// TwinCAT 3 PLC project PLC
// ProgramVersion: 3.1.4026.13
// libraries:
//   Tc2_Standard, * (Beckhoff Automation GmbH)
//   Tc2_System, * (Beckhoff Automation GmbH)
//   Tc3_Module, * (Beckhoff Automation GmbH)
// project tree:
//   Control/ FB_ControlSignal.TcPOU, FB_FeedForward.TcPOU, FB_PID.TcPOU (not stored), FB_Running.TcPOU (not stored), G_Mode.TcGVL
//   Filtering/ FB_Filtering.TcPOU (not stored), G_Filtered.TcGVL (not stored)
//   GVL/ G_Enables.TcGVL (not stored), G_FilterConstants.TcGVL (not stored), G_OPC.TcGVL, G_Parameter.TcGVL
//   Inputs/Function Blocks/ FB_FlowTransform.TcPOU, FB_JoystickInputScaling.TcPOU, FB_Normalize.TcPOU (not stored), FB_Normalize_Joystick.TcPOU, FB_PositionInputScaling.TcPOU (not stored)
//   Inputs/ G_Inputs.TcGVL
//   MotionRef/ FB_AutoClock.TcPOU (not stored), FB_DeadbandTester.TcPOU, FB_InitialPos.TcPOU (not stored), FB_MotionRef.TcPOU, FB_RunClock.TcPOU (not stored)
//   Outputs/ FB_ValveOutput.TcPOU (not stored), G_Output.TcGVL (not stored)
//   / PlcTask.TcTTO (not stored)
//   Programs/ MAIN.TcPOU (not stored), P_ControlBlock.TcPOU, P_FeedForward.TcPOU (not stored), P_Filtering.TcPOU (not stored), P_Inputs.TcPOU, P_Modes.TcPOU (not stored), P_Output.TcPOU (not stored), P_PID.TcPOU (not stored), P_RunClock.TcPOU (not stored)
//   XML/ FB_Derivator.TcPOU (not stored), FB_Integrator.TcPOU (not stored), G_Init.TcGVL (not stored)
// real-time tasks:
//   TASK PlcTask: cycle T#1ms, priority 20, ADS port 350
// I/O:
//   DEVICE Device 4 (EtherCAT), AmsNetId 5.107.189.26.5.1
//     RIO (EK1100) [EK1100 EtherCAT Coupler (2A E-Bus)]
//       DI (EL1008) [EL1008 8Ch. Dig. Input 24V, 3ms]
//       DO (EL2008) [EL2008 8Ch. Dig. Output 24V, 0.5A]
//       AI1 (EL3068) [EL3068 8Ch. Ana. Input 0-10V]
//       AI2 (EL3068) [EL3068 8Ch. Ana. Input 0-10V]
//       AI3 (EL3174) [EL3174 4Ch. Ana. Input +/-10V Diff., +/-20mA SingleEnded, 16 Bit]
//       AO (EL4104) [EL4104 4Ch. Ana. Output 0-10V, 16bit]
//       End Cap (EL9011) [EL9011 End Terminal]
// variable links:
//   PLC/PLC Instance <-> Device 4 (EtherCAT)/RIO (EK1100)/AI1 (EL3068)
//     PlcTask Inputs/G_Inputs.nRawJoystick <-> AI Standard Channel 2/Value
//     PlcTask Inputs/G_Inputs.nRawPistonPosition <-> AI Standard Channel 3/Value
//   PLC/PLC Instance <-> Device 4 (EtherCAT)/RIO (EK1100)/AI2 (EL3068)
//     PlcTask Inputs/G_Inputs.nRawPa <-> AI Standard Channel 4/Value
//     PlcTask Inputs/G_Inputs.nRawPaLower <-> AI Standard Channel 5/Value
//     PlcTask Inputs/G_Inputs.nRawPb <-> AI Standard Channel 6/Value
//     PlcTask Inputs/G_Inputs.nRawPs <-> AI Standard Channel 1/Value
//   PLC/PLC Instance <-> Device 4 (EtherCAT)/RIO (EK1100)/AI3 (EL3174)
//     PlcTask Inputs/G_Inputs.nRawFlow <-> AI Standard Channel 1/Value
//   PLC/PLC Instance <-> Device 4 (EtherCAT)/RIO (EK1100)/AO (EL4104)
//     PlcTask Outputs/G_Output.nValveOutput <-> AO Output Channel 1/Analog output
//   PLC/PLC Instance <-> Device 4 (EtherCAT)/RIO (EK1100)/DI (EL1008)
//     PlcTask Inputs/G_Inputs.bAuto <-> Channel 1/Input
//     PlcTask Inputs/G_Inputs.bManual <-> Channel 2/Input
//     PlcTask Inputs/G_Inputs.bStartButton <-> Channel 3/Input
//     PlcTask Inputs/G_Inputs.bStopButton <-> Channel 4/Input
//   PLC/PLC Instance <-> Device 4 (EtherCAT)/RIO (EK1100)/DO (EL2008)
//     PlcTask Outputs/G_Output.bGreenLight <-> Channel 1/Output
//     PlcTask Outputs/G_Output.bRedLight <-> Channel 2/Output
//     PlcTask Outputs/G_Output.bRunning <-> Channel 3/Output

// ---- Control/G_Mode.TcGVL
{attribute 'qualified_only'}
VAR_GLOBAL
	bRunning : BOOL;
	bManual : BOOL;
	bAuto : BOOL;
END_VAR

// ---- GVL/G_OPC.TcGVL
{attribute 'qualified_only'}
VAR_GLOBAL
	
	// Unfiltered Pressures
	fPa : LREAL;
	fPb : LREAL;
	fPs : LREAL;
	fPaLower : LREAL;
	
	// Filtered Pressures
	fPaFiltered : LREAL;
	fPbFiltered : LREAL;
	fPsFiltered : LREAL;
	fPaLowerFiltered : LREAL;
	
	
	fPistonPosition : LREAL;
	fJoystick : LREAL;
	fFlow : LREAL;
	fFlowBit : LREAL;
	
	fXRef : LREAL;
	fXDotRef : LREAL;
	
	fU : LREAL;
	fTime : LREAL;
	fError : LREAL;
	fSignalPID : LREAL;
	fUFF : LREAL;
END_VAR

// ---- GVL/G_Parameter.TcGVL
{attribute 'qualified_only'}
VAR_GLOBAL
	// Motion Ref
	fAmplitude : LREAL := 0.1;
	fMean : LREAL := 0.2;
	fFrequency : LREAL := 0.05;
	
	fQMaxDown : LREAL := 15.9;
	fQMaxUp : LREAL := 24.4;
	fDeadUp : LREAL := 0.13;
	fDeadDown : LREAL := 0.12;
	
	// Deadband test
	fConst : LREAL := 0.0; // [-1, 1]

	
	fCycleTime : LREAL := 0.001; // Time Step [s]
	fQConst : LREAL := 15;
	
	// PID-constants
	Kp 	: LREAL := 7.0; // P
	Ki 	: LREAL := 0.0;	// I
	Kd 	: LREAL := 0.0;	// D
	KFF : LREAL := 0.85; // Coefficient of FeedForward
	
END_VAR

// ---- Inputs/G_Inputs.TcGVL
{attribute 'qualified_only'}
VAR_GLOBAL
	// Mode Selector
	bManual 			AT %I* : BOOL;
	bAuto	 			AT %I* : BOOL;
	bStartButton		AT %I* : BOOL;
	bStopButton			AT %I* : BOOL;
	
	// Raw Pressure Values
	nRawPa 				AT %I*	: INT;
	nRawPb				AT %I*	: INT;
	nRawPs				AT %I*	: INT;
	nRawPaLower			AT %I* 	: INT;
	
	// Raw Position Values
	nRawPistonPosition 	AT %I*	: INT;
	nRawJoystick		AT %I*	: INT;
	nRawFlow			AT %I*	: INT; // [-150, 150]
END_VAR

// ---- Control/FB_ControlSignal.TcPOU
FUNCTION_BLOCK FB_ControlSignal
VAR_INPUT
	fUFF : LREAL;
	fPID : LREAL;
	bEnableU : BOOL;
	fQMaxUp 	: LREAL; // Needs to be positive (22)
	fQMaxDown 	: LREAL; // Needs to be positive (15)
	fDeadUp		: LREAL; // Needs to be positive (0.155)
	fDeadDown 	: LREAL; // Needs to be positive (0.18)
	
	fXDotRef	: LREAL;
	fError		: LREAL;
END_VAR
VAR_OUTPUT
	fU : LREAL;
END_VAR
VAR

	fUTemp : LREAL;
	fUTemp2 : LREAL;
	fUMax : LREAL := 0.9;
END_VAR

IF bEnableU THEN
	fUTemp := fUFF  - fPID;
	
	// Deadband compensation
	IF (fXDotRef > 0 OR fXDotRef < 0) OR fError > 0.002 THEN
		IF fUTemp <= 0.0 THEN	// Upwards
			fUTemp2 := fUTemp - fDeadUp;
		ELSIF fUTemp > 0.0 THEN // Downwards
			fUTemp2 := fUTemp + fDeadDown;
		END_IF
		
		IF fUTemp2 >= fUMax THEN
			fU := fUMax;
		ELSIF fUTemp2 <= -fUMax THEN
			fU := -fUMax;
		ELSE
			fU := fUTemp2;
		END_IF
	ELSE
		fU := 0.0;
	END_IF
END_IF

END_FUNCTION_BLOCK

// ---- Control/FB_FeedForward.TcPOU
FUNCTION_BLOCK FB_FeedForward
VAR_INPUT
	fXDotRef 	: LREAL; // Motion Referance
	fQMaxUp 	: LREAL; // Needs to be positive (22)
	fQMaxDown 	: LREAL; // Needs to be positive (15)
	fDeadUp		: LREAL; // Needs to be positive (0.155)
	fDeadDown 	: LREAL; // Needs to be positive (0.18)
	fPs 		: LREAL;
	fPa			: LREAL;
	fPb			: LREAL;
	fKFF 		: LREAL; // Coefficient of FeedForward
END_VAR
VAR_OUTPUT
	fUFF : LREAL;
END_VAR
VAR
	fUTemp : LREAL;
	fUMax : LREAL := 0.9;
	fQRef : LREAL;
	fAp : LREAL := 33.1 / 10000.0;
	fAa : LREAL := 23.56 / 10000.0;
	
	fK02Up : LREAL := 0.78; //0.78;
	fK04Up : LREAL := 2.29; //2.3;
	fK06Up : LREAL := 3.42;// 3.27;
	fK07Up : LREAL := 4.59; //4.54;
	fK08Up : LREAL := 5.09; //4.94;
	fK1Up : LREAL := 5.71; //5.68;
	
	fK02Down : LREAL := -0.75; //-0.75; 
	fK04Down : LREAL := -2.17; //-2.21; //-1.37;
	fK06Down : LREAL := -3.39; //-3.45; 
	fK07Down : LREAL := -3.99; //-3.96; //-2.45;
	fK08Down : LREAL := -4.55; //-4.61; 
	fK1Down : LREAL := -4.84; //-4.67; //-2.88;
	
	fDeltaP : LREAL;
	fKRef : LREAL; 
	
END_VAR



IF fXDotRef >= 0.0 THEN // Upwards
	
	fQRef := fAp * fXDotRef * 60000;
	fDeltaP := fPs - fPa;
	IF fDeltaP < 100 THEN
		fDeltaP := 100;
	ELSE
		fDeltaP := fDeltaP;
	END_IF
	fKRef := fQRef / SQRT(fDeltaP);
	
	IF fKRef < 0.0 THEN
		fUTemp := 0.0;
	ELSIF fKRef < fK02Up THEN
		fUTemp := -fKRef/fK02Up * (0.2 - fDeadUp);
	ELSIF fKRef < fK04Up THEN
		fUTemp := -(0.2 - fDeadUp) -(fKRef - fK02Up) / (fK04Up - fK02Up) * (0.4-fDeadUp-0.2);
	ELSIF fKRef < fK06Up THEN
		fUTemp := -(0.4 - fDeadUp - 0.2) - (0.2 - fDeadUp) - (fKRef - fK04Up) / (fK06Up - fK04Up) * (0.6-fDeadUp-0.4);
	ELSIF fKRef < fK07Up THEN
		fUTemp := -(0.6 - fDeadUp - 0.4) - (0.4 - fDeadUp - 0.2) - (0.2 - fDeadUp) - (fKRef - fK06Up) / (fK07Up - fK06Up) * (0.7 - fDeadUp - 0.6);
	ELSIF fKRef < fK08Up THEN
		fUTemp := -(0.7 - fDeadUp - 0.6) - (0.6 - fDeadUp - 0.4) - (0.4 - fDeadUp - 0.2 ) - (0.2 - fDeadUp) - (fKRef - fK07Up) / (fK08Up - fK07Up) * (0.8-fDeadUp-0.7);
	ELSIF fKRef < fK1Up THEN
		fUTemp := -(0.8 - fDeadUp - 0.7) - (0.7 - fDeadUp - 0.6) - (0.6 - fDeadUp - 0.4) - (0.4 - fDeadUp - 0.2 ) - (0.2 - fDeadUp) - (fKRef - fK08Up) / (fK1Up - fK08Up) * (1.0-fDeadUp-0.8);
	ELSE
		fUTemp := -(1 - fDeadUp);
	END_IF
	
//	fUTemp := -((fQRef/fQMaxUp) * (fUMax-fDeadUp));

ELSIF fXDotRef < 0.0 THEN // Downwards
	
	fQRef := fAa * fXDotRef * 60000;
	fDeltaP := fPs - fPb;
	IF fDeltaP < 100 THEN
		fDeltaP := 100;
	ELSE
		fDeltaP := fDeltaP;
	END_IF
	fKRef := fQRef / SQRT(fDeltaP);
	
	IF fKRef > 0.0 THEN
		fUTemp := 0.0;
	ELSIF fKRef > fK02Down THEN
		fUTemp := fKRef/fK02Down * (0.2-fDeadDown);
	ELSIF fKRef > fK04Down THEN
		fUTemp := (0.2 - fDeadDown) + (fKRef - fK02Down) / (fK04Down - fK02Down) * (0.4 - fDeadDown - 0.2);
	ELSIF fKRef > fK06Down THEN
		fUTemp := (0.2 - fDeadDown) + (0.4 - fDeadDown) + (fKRef - fK04Down) / (fK06Down - fK04Down) * (0.6 - fDeadDown - 0.4);
	ELSIF fKRef > fK07Down THEN
		fUTemp := (0.2 - fDeadDown) + (0.4 - fDeadDown) + (0.6 - fDeadDown) + (fKRef - fK06Down) / (fK07Down - fK06Down) * (0.7 - fDeadDown - 0.6);
	ELSIF fKRef > fK08Down THEN
		fUTemp := (0.2 - fDeadDown) + (0.4 - fDeadDown) + (0.6 - fDeadDown) + (0.7 - fDeadDown) + (fKRef - fK07Down) / (fK08Down - fK07Down) * (0.8 - fDeadDown - 0.7);
	ELSIF fKRef > fK1Down THEN
		fUTemp := (0.2 - fDeadDown) + (0.4 - fDeadDown) + (0.6 - fDeadDown) + (0.7 - fDeadDown) + (0.8 - fDeadDown) + (fKRef - fK08Down) / (fK1Down - fK08Down) * (1.0 - fDeadDown - 0.8);
	ELSE
		fUTemp := (1.0 - fDeadDown);
	END_IF
	
//	fUTemp := -((fQRef/fQMaxDown) * (fUMax-fDeadDown)); // FDeadDown needs to be positive
	

END_IF

fUFF := fUTemp * fKFF; // Tomec

END_FUNCTION_BLOCK

// ---- Inputs/Function Blocks/FB_FlowTransform.TcPOU
FUNCTION_BLOCK FB_FlowTransform
VAR_INPUT
	bEnable : BOOL;
	nRawInput : INT;
END_VAR
VAR_OUTPUT
	fOutput : LREAL;
	fOutputBit : LREAL;
END_VAR
VAR
	fRawInput : LREAL;
	fTempInput : LREAL;
	fTempOutput : LREAL;
	fMaxInputValue			: LREAL := 32767.0;
	fNeutralInputValue  	: LREAL := 15250.0;
	fMinInputValue 			: LREAL := 0.0;
	
	fNeutralDeadband		: LREAL := 25.0;
	
	fMaxOutputValue  		: LREAL := 150.0;
	fNeutralOutputValue  	: LREAL := 0.0;
	fMinOutputValue  		: LREAL := -150.0;
	
END_VAR

fRawInput := INT_TO_LREAL(nRawInput);

fTempInput := fRawInput - fNeutralInputValue;

IF fTempInput > fNeutralDeadband THEN
	fTempOutput := fMaxOutputValue * fTempInput/(fMaxInputValue - fNeutralInputValue);
ELSIF fTempInput < -fNeutralDeadband THEN	
	fTempOutput := fMinOutputValue * (fTempInput)/(fNeutralInputValue - fMinInputValue);
ELSE
	fTempOutput := 0.0;
END_IF

IF NOT(bEnable) THEN
	fOutput := 0.0;
ELSE
	fOutput := LIMIT(fMinOutputValue, fTempOutput, fMaxOutputValue);
END_IF

fOutputBit := INT_TO_LREAL(nRawInput);

END_FUNCTION_BLOCK

// ---- Inputs/Function Blocks/FB_JoystickInputScaling.TcPOU
FUNCTION_BLOCK FB_JoystickInputScaling
VAR_INPUT
	bEnable : BOOL;
	nRawInput : INT;
END_VAR
VAR_OUTPUT
	fOutput : LREAL;
END_VAR
VAR
	fRawInput : LREAL;
	fTempInput : LREAL;
	fTempOutput : LREAL;
	fMaxInputValue			: LREAL := 14746.0;
	fMinInputValue 			: LREAL := 1617.0;
	fNeutralInputValue  	: LREAL := 8160.0;
	fNeutralDeadband		: LREAL := 50.0;
	fMaxOutputValue  		: LREAL := 1.0;
	fMinOutputValue  		: LREAL := -1.0;
	fNeutralOutputValue  	: LREAL := 0.0;
END_VAR

fRawInput := INT_TO_LREAL(nRawInput);

fTempInput := fRawInput - fNeutralInputValue;

IF fTempInput > fNeutralDeadband THEN
	fTempOutput := fTempInput/(fMaxInputValue - fNeutralInputValue);
ELSIF fTempInput < -fNeutralDeadband THEN	
	fTempOutput := fTempInput/(fNeutralInputValue - fMinInputValue);
ELSE
	fTempOutput := 0.0;
END_IF

IF NOT(bEnable) THEN
	fOutput := 0.0;
ELSE
	fOutput := LIMIT(fMinOutputValue, fTempOutput, fMaxOutputValue);
END_IF

END_FUNCTION_BLOCK

// ---- Inputs/Function Blocks/FB_Normalize_Joystick.TcPOU
FUNCTION_BLOCK FB_Normalize_Joystick
VAR_INPUT
	nRawInput : INT;
	fMaxSignal : LREAL;
	fMinSignal : LREAL;
END_VAR
VAR_OUTPUT
	fNormalizedInput : LREAL;
END_VAR
VAR
END_VAR

fNormalizedInput := (INT_TO_LREAL(nRawInput) - 32767.0/2.0) / (32767.0/2.0);

fNormalizedInput := LIMIT(fMinSignal,fNormalizedInput,fMaxSignal);

END_FUNCTION_BLOCK

// ---- MotionRef/FB_DeadbandTester.TcPOU
FUNCTION_BLOCK FB_DeadbandTester
VAR_INPUT
	fInput : LREAL;
	bEnable : BOOL;
	fConst : LREAL;
END_VAR
VAR_OUTPUT
	fOutput : LREAL;
	fXDotRef : LREAL;
END_VAR
VAR
	
END_VAR

IF bEnable THEN
	fOutput := fInput;
ELSE
	fOutput := fConst;
	fXDotRef := 0.0000001;
END_IF

END_FUNCTION_BLOCK

// ---- MotionRef/FB_MotionRef.TcPOU
FUNCTION_BLOCK FB_MotionRef
VAR_INPUT
	fTime : LREAL;
	fAmplitude : LREAL;
	fFrequency : LREAL;
	fInitialPos : LREAL;
END_VAR
VAR_OUTPUT
	fXDotRef : LREAL;
	fXRef : LREAL;
END_VAR
VAR
	fPI : LREAL := 3.1415;
	fMean : LREAL;
END_VAR

fMean := fAmplitude + fInitialPos; 
IF G_Inputs.bStartButton THEN
	fXRef := fMean - fAmplitude * COS(2*fPI * fFrequency * fTime);
	fXDotRef := 2 * fPI *fFrequency * fAmplitude * SIN(2*fPI * fFrequency * fTime);
ELSE
	fXDotRef := 0.0;
END_IF

END_FUNCTION_BLOCK

// ---- Programs/P_ControlBlock.TcPOU
PROGRAM P_ControlBlock
VAR
	fbDeadBandTester : FB_DeadbandTester;
	fbAutoClock : FB_AutoClock;
	fbMotionRef : FB_MotionRef;
	fbControl : FB_ControlSignal;
	fbInitialPos : FB_InitialPos;
END_VAR


fbInitialPos(
	bEnable := G_Mode.bRunning,
	fCurrentPos := G_OPC.fPistonPosition
);

fbMotionRef(
	fInitialPos := fbInitialPos.fInitialPos
);

IF G_Mode.bAuto AND G_Mode.bRunning THEN
	


fbAutoClock(
	fStart := G_Inputs.bStartButton,
	fRunning := G_Mode.bRunning,
	fCycle := G_Parameter.fCycleTime
);

fbMotionRef(
	fTime := fbAutoClock.fTime,
	fAmplitude := G_Parameter.fAmplitude,
	fInitialPos := fbInitialPos.fInitialPos,
	fFrequency := G_Parameter.fFrequency,
	fXDotRef => G_OPC.fXDotRef,
	fXRef => G_OPC.fXRef 
);

fbControl(
	fUFF := G_OPC.fUFF,
	fPID := G_OPC.fSignalPID,
	bEnableU := G_Enables.bEnableU,
	fQMaxUp := G_Parameter.fQMaxUp,
	fQMaxDown := G_Parameter.fQMaxDown,
	fDeadUp := G_Parameter.fDeadUp,
	fDeadDown := G_Parameter.fDeadDown,
	fXDotRef := G_OPC.fXDotRef,
	fError := G_OPC.fError,
	
	fU => G_OPC.fU
);

ELSIF G_Mode.bManual AND G_Mode.bRunning THEN

fbInitialPos(
	bEnable := G_Inputs.bStartButton,
	fCurrentPos := G_OPC.fPistonPosition
);
fbDeadBandTester(
	fInput := G_OPC.fJoystick,
	bEnable := G_Enables.bDeadBandTest,
	fConst := G_Parameter.fConst,
	fOutput => G_OPC.fU,
	fXDotRef => G_OPC.fXDotRef
);

END_IF

END_PROGRAM

// ---- Programs/P_Inputs.TcPOU
PROGRAM P_Inputs
VAR
	fbNormPa :  FB_Normalize;
	fbNormPb :  FB_Normalize;
	fbNormPs :  FB_Normalize;
	fbNormPaLower : FB_Normalize;
	
	fbNormPistonPosition : FB_PositionInputScaling;
	fbJoystick : FB_JoystickInputScaling;
	fbFlow : FB_FlowTransform;

	fPa : LREAL;
	fPb : LREAL;
	fPs : LREAL;
	fPaLower : LREAL;
	
	fPistonPosition : LREAL;
END_VAR

fbNormPa(
	nRawInput := G_Inputs.nRawPa,
	fMaxValue := 400.0, 			// [Bar]
	fNormalizedInput => G_OPC.fPa
);

fbNormPb(
	nRawInput := G_Inputs.nRawPb,
	fMaxValue := 400.0, 			// [Bar]
	fNormalizedInput => G_OPC.fPb
);

fbNormPs(
	nRawInput := G_Inputs.nRawPs,
	fMaxValue := 400.0, 			// [Bar]
	fNormalizedInput => G_OPC.fPs
);

fbNormPistonPosition(
	nRawInput := G_Inputs.nRawPistonPosition,
	fOutput => G_OPC.fPistonPosition
);
	
fbJoystick(
	nRawInput := G_Inputs.nRawJoystick,
	bEnable := (G_Mode.bRunning AND G_Mode.bManual),
	fOutput => G_OPC.fJoystick
);

fbNormPaLower(
	nRawInput := G_Inputs.nRawPaLower,
	fMaxValue := 400.0, 			// [Bar]
	fNormalizedInput => G_OPC.fPaLower
);

fbFlow(
	nRawInput := G_Inputs.nRawFlow,
	bEnable := TRUE,
	fOutput => G_OPC.fFlow,
	fOutputBit => G_OPC.fFlowBit
);

END_PROGRAM
